{attribute 'qualified_only'}
{attribute 'strict'}
TYPE MoverDirection_e :
(
	Farward,
	Reverse
);
END_TYPE

(* stored: Version 1.1.0.1, ProductVersion 3.1.4024.6
   EnumerationTextList MoverDirection_e: Id {662e428d-8bd9-412a-a595-5e82fe2435cd} *)
